PROGRAM posCarrinho
VAR
	timeCalc: TIME;
	bNotificaTime: BOOL:= TRUE;
END_VAR


///// CALCULO DE DEFINIÇÃO SE O PROCESSO PASSA DAS 36 HORAS LIMITES ----------------------------------------
timeCalc:= (gvl_p.arrStatusEstufas[0].prevFimSeca - systemtime_to_dt(gvl.fbGetLocalSystemTime.systemTime));
IF timeCalc < T#24H THEN
	bNotificaTime:= FALSE;
	ELSE
		bNotificaTime:= TRUE;
		
END_IF

END_PROGRAM

(* stored: Version 1.1.0.1, ProductVersion 3.1.4024.12
   POU posCarrinho: Id {846c8a73-d440-42fe-a20b-dd688f0ae5ff}, SpecialFunc None *)
